(* CoDeSys 2.3 export: SELECTORCLASS.EXP *)

(* Data type in ENUM *)
TYPE SelectorClass : (ReversiveTransport:=1, TwoStage, MultiStage);
END_TYPE
